INTERFACE I_StateList

METHOD AddStateAtIndex
VAR_INPUT
	Index : DINT;
	State : I_State;
END_VAR
END_METHOD

METHOD GetStateAtIndex : I_State
VAR_INPUT
	Index : DINT;
END_VAR
END_METHOD

PROPERTY NumberOfStates : DINT
GET
END_GET
END_PROPERTY

END_INTERFACE

(* stored: Version 1.1.0.1, ProductVersion 3.1.4026.18
   Itf I_StateList: Id {60804661-a2c8-4da3-98f9-b20e61cb1ed4}
   Method AddStateAtIndex: Id {90d469bb-6b8d-4455-8cf4-5e391435322d}
   Method GetStateAtIndex: Id {8aa82c5b-d67f-49f6-9ab0-14175bede0d0}
   Property NumberOfStates: Id {e3baf465-ff88-4c73-b9d9-3325dbcbdf9f}
   Get Get: Id {3879470a-1b4e-4083-a471-79c21b07cf07} *)
